// TIA Portal V19 export
FUNCTION_BLOCK "TYPIC_C401_BF_RSS"   // FB105, FBD
TITLE = TYPIC_C401_BF_RSS: Rijstrooksignalisatie
{ S7_Optimized_Access := 'TRUE' }
AUTHOR : OCOTECH
FAMILY : Typical
NAME : C401.801
// Logisch Object Besturing: C401.801
// 
// De basisfunctie Rijstrooksignalisatie maakt een algemene status aan van de rijstrooksignalisatie voor een verkeerskoker.
// stored: MemoryReserve 10, SetENOAutomatically false
   VAR_INPUT
      CFG_MAX_NOK1 { ExternalAccessible := 'False'; ExternalVisible := 'False'; ExternalWritable := 'False'} : Int;   // Maximum aantal niet observeerbare RSS-borden ter voorkoming beschikbaarheidsstatus niet beschikbaar
      CFG_MAX_NOK2 { ExternalAccessible := 'False'; ExternalVisible := 'False'; ExternalWritable := 'False'} : Int;   // Maximum aantal opeenvolgende niet observeerbare RSS-borden per rijstrook ter voorkoming beschikbaarheidsstatus niet beschikbaar
      STU_ALG_LCK_SIG { ExternalAccessible := 'False'; ExternalVisible := 'False'; ExternalWritable := 'False'} : USInt;   // Onderdruk alarmen
   END_VAR
   VAR_IN_OUT
      VAR_RSS : Array[*] of "C401_VAR_RSS_TYPIC";   // Array van alle RSS-borden met een struct met alle variabelen van het RSS-bord
   END_VAR
   VAR
      SIG { ExternalWritable := 'False'} : Struct   // Signaleringen
         AB01 : Bool;   // Rijstrook signalisatie beperkt beschikbaar
         AB02 : Bool;   // Rijstrook signalisatie niet beschikbaar
      END_STRUCT;
      VAR { ExternalWritable := 'False'} : Struct   // Variabelen
         BSC : USInt;   // Geeft de beschikbaarheid aan van het rijstrooksignalisatie
         VGV_SIG_VOP : Bool;   // TRUE = Signaleringen vrijgegeven voor verkeersoperator FALSE = Onderdrukt
         AANT_NOK { ExternalAccessible := 'False'; ExternalVisible := 'False'} : USInt;   // Totaal aantal niet observeerbare RSS-borden
         MAX_NOK { ExternalAccessible := 'False'; ExternalVisible := 'False'} : USInt;   // Maximum gedetecteerd aantal opeenvolgende niet observeerbare RSS-borden per rijstrook
         HULP_NOK { ExternalAccessible := 'False'; ExternalVisible := 'False'} : USInt;   // Hulpvariabele voor maximum gedetecteerd aantal opeenvolgende niet observeerbare RSS-borden per rijstrook
         LUS_STO { ExternalAccessible := 'False'; ExternalVisible := 'False'} : USInt;   // OK = geen enkel luspaar geeft FOUT FOUT = een of meer lusparen geeft FOUT
      END_STRUCT;
   END_VAR
BEGIN

REGION Network 1: START
END_REGION

REGION Network 2: +++ Niet observeerbare RSS-borden en vaststelling luspaar storing +++
   // Deze functie omvat het tellen van het aantal RSS-borden dat niet observeerbaar is, tellen van het maximum aantal opeenvolgende RSS-borden dat niet observeerbaar is over een rijstrook en het vaststellen of er een luspaar een storing heeft.
END_REGION

REGION Network 3: +++ Bepalen beschikbaarheidsstatus +++
   // Beschikbaarheidsstatus (beschikbaar / beperkt beschikbaar / niet beschikbaar) bepalen.
END_REGION

REGION Network 4 (SCL): Beschikbaarheidsstatus bepalen
   IF 
       //voorwaarden "Niet beschikbaar"
       TRUE
   THEN
       //Beschikbaarheidsstatus = Niet Beschikbaar
       #VAR.BSC:= "NietBeschikbaar";
   ELSIF
       //voorwaarden "Beperkt beschikbaar"
       TRUE
   THEN
       //Beschikbaarheidsstatus = Beperkt Beschikbaar
       #VAR.BSC:= "Beperkt";
   ELSE
       //Beschikbaarheidsstatus = Beschikbaar
       #VAR.BSC:= "Beschikbaar";
   END_IF;
END_REGION

REGION Network 5: +++ Signaleringen +++
   // Aanmaken signaleringen.
END_REGION

REGION Network 6: Signalering AB01 : Niet Beschikbaar
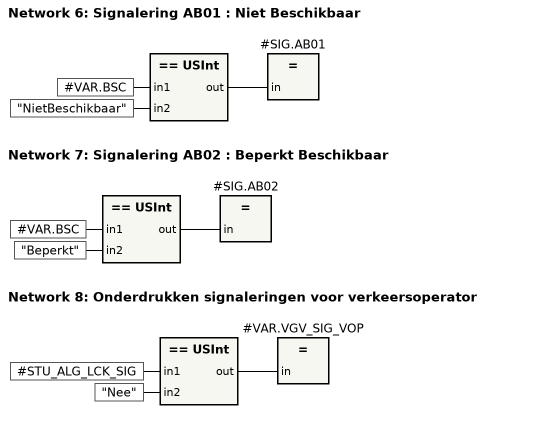
   #SIG.AB01 := #VAR.BSC = "NietBeschikbaar";
END_REGION

REGION Network 7: Signalering AB02 : Beperkt Beschikbaar
   #SIG.AB02 := #VAR.BSC = "Beperkt";
END_REGION

REGION Network 8: Onderdrukken signaleringen voor verkeersoperator
   // Via de variabele VGV_SIG_VOP wordt aan IRIS SCADA doorgegeven of signaleringen (bestemd voor de verkeersoperator) van de deze functie zichtbaar (of onderdrukt) moeten zijn.
   #VAR.VGV_SIG_VOP := #STU_ALG_LCK_SIG = "Nee";
END_REGION

REGION Network 9: EINDE
   // Variabelen van intern scada rakvlak naar outputs copieren
END_REGION
END_FUNCTION_BLOCK
